% RSLogix 500 project I2P JOB 07 - MYAH.RSS, saved by version 10.00.00.00 %
PROJECT "ML05B"    % processor: Bul.1763 MicroLogix 1100 Series B %

PROGRAM FILES
  LAD 2   3 rungs

DATA FILES
  O0 OUTPUT  4 elements
  I1 INPUT  6 elements
  S2 STATUS  66 elements
  B3 BINARY  1 elements
  T4 TIMER  1 elements
  C5 COUNTER  1 elements
  R6 CONTROL  1 elements
  N7 INTEGER  1 elements
  F8 FLOAT  1 elements

LADDER 2
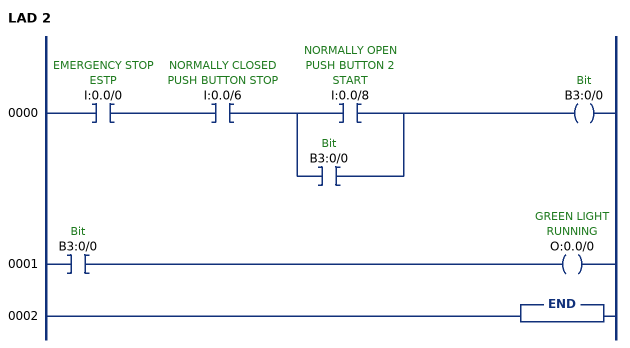
% Rung: 0 %
SOR XIC I:0.0/0 XIC I:0.0/6 BST XIC I:0.0/8 NXB XIC B3:0/0 BND OTE B3:0/0 EOR
%   I:0.0/0  ESTP  "EMERGENCY STOP" %
%   I:0.0/6  STOP  "NORMALLY CLOSED PUSH BUTTON" %
%   I:0.0/8  START  "NORMALLY OPEN PUSH BUTTON 2" %
%   B3:0/0  "Bit" %
% Rung: 1 %
SOR XIC B3:0/0 OTE O:0.0/0 EOR
%   B3:0/0  "Bit" %
%   O:0.0/0  RUNNING  "GREEN LIGHT" %
% Rung: 2 %
SOR END EOR

OTHER DOCUMENTED ADDRESSES
  I:0.0/1  CR1_CON  "CONTROL RELAY 1 CONTACT"
  I:0.0/2  CR2_CON  "CONTROL RELAY 2 CON"
  I:0.0/3  3PSS_A  "3 POSITION SELCTOR SWITCH A POSITION"
  I:0.0/4  3PSS_B  "3 POSITION SELECTOR SWITCH B POSITON"
  I:0.0/5  2PSS  "2 POSITION SELECTOR SWITCH"
  I:0.0/7  NO_PB1  "NORMALLY OPEN PUSH BUTTON 1"
  O:0.0/1  YLW_LT  "YELLOW LIGHT"
  O:0.0/2  RED_LT  "RED LIGHT"
  O:0.0/3  BLU_LT  "BLUE LIGHT"
  O:0.0/4  CR1  "CONTROL RELAY 1"
  O:0.0/5  CR2  "CONTROL RELAY 2"
